// TwinCAT 3 PLC project SmartLiquidFillingSystem
// ProgramVersion: 3.1.4024.0
// libraries:
//   Tc2_Standard, * (Beckhoff Automation GmbH)
//   Tc2_System, * (Beckhoff Automation GmbH)
//   Tc3_Module, * (Beckhoff Automation GmbH)
// project tree:
//   DUTs/ E_LiquidType.TcDUT, E_StationState.TcDUT, ST_Bottle.TcDUT
//   GVLs/ GVL_References.TcGVL
//   / PlcTask.TcTTO
//   POUs/ FB_HoneyFill.TcPOU, FB_SodaFill.TcPOU, FB_StationController.TcPOU, FB_WaterFill.TcPOU, F_StrategyFunction.TcPOU, I_FillingStrategy.TcIO, MAIN.TcPOU
// (motion and I/O tree: see PLC project instructions_practice)
// real-time tasks:
//   TASK PlcTask: cycle T#10ms, priority 20, ADS port 350
//   TASK PlcTask1: cycle T#10ms, priority 22, ADS port 351
//   TASK PlcTask2: cycle T#10ms, priority 21, ADS port 352
//   TASK PlcTask3: cycle T#10ms, priority 23, ADS port 353

CONFIGURATION SmartLiquidFillingSystem
    RESOURCE PLC ON TwinCAT3
        TASK PlcTask(INTERVAL := T#10ms, PRIORITY := 23);
        PROGRAM MAIN WITH PlcTask : MAIN;
    END_RESOURCE
END_CONFIGURATION

// ---- DUTs/E_LiquidType.TcDUT
{attribute 'qualified_only'}
{attribute 'strict'}
TYPE E_LiquidType :
(
	WATER := 0,
	HONEY,
	SODA
);
END_TYPE

// ---- DUTs/E_StationState.TcDUT
{attribute 'qualified_only'}
{attribute 'strict'}
TYPE E_StationState :
(
	IDLE := 0,
	DETECTION,
	FILLING,
	COMPLETE,
	ERROR
);
END_TYPE

// ---- DUTs/ST_Bottle.TcDUT
TYPE ST_Bottle :
STRUCT
	nId  : DINT ;
	fCurrentLevel : REAL;
	fTargetLevel : REAL;
	eLiquidType : E_LiquidType;
END_STRUCT
END_TYPE

// ---- GVLs/GVL_References.TcGVL
{attribute 'qualified_only'}
VAR_GLOBAL
    g_fbHoneyFill : FB_HoneyFill;
    g_fbSodaFill  : FB_SodaFill;
    g_fbWaterFill : FB_WaterFill;
END_VAR

// ---- POUs/I_FillingStrategy.TcIO
INTERFACE I_FillingStrategy

METHOD ExecuteFill : BOOL
VAR_INPUT
	stBottle : REFERENCE TO ST_Bottle;
END_VAR
END_METHOD

END_INTERFACE

// ---- POUs/MAIN.TcPOU
PROGRAM MAIN
VAR
	bStart : BOOL;
	
	stBottle1 : ST_Bottle := (nId := 101, fTargetLevel := 70, eLiquidType := E_LiquidType.HONEY);
	stBottle2 : ST_Bottle := (nId := 102, fTargetLevel := 85, eLiquidType := E_LiquidType.SODA);
	stBottle3 : ST_Bottle := (nId := 103, fTargetLevel := 90, eLiquidType := E_LiquidType.WATER);
	
	
	fbStationController1 : FB_StationController;
	fbStationController2: FB_StationController;
	fbStationController3 : FB_StationController;
	
	
END_VAR

IF bStart THEN
	fbStationController1(stBottle := stBottle1);
	fbStationController2(stBottle := stBottle2);
	fbStationController3(stBottle := stBottle3);
	bStart := FALSE;
END_IF

END_PROGRAM

// ---- POUs/FB_StationController.TcPOU
FUNCTION_BLOCK FB_StationController

VAR_IN_OUT
	stBottle : ST_Bottle;
END_VAR
VAR
	iFillingStrategy : I_FillingStrategy;
	eStationState : E_StationState;
	nCompleteCount : DINT;
	nDefectCount : DINT;
END_VAR

IF  __ISVALIDREF(stBottle) THEN
	CASE eStationState OF
	E_StationState.IDLE:
		eStationState := E_StationState.DETECTION;
	
	E_StationState.DETECTION:
	iFillingStrategy := F_StrategyFunction(stBottle);
	IF iFillingStrategy <> 0 THEN
		eStationState := E_StationState.FILLING;
	ELSE
		eStationState := E_StationState.ERROR;
	END_IF
	
	E_StationState.FILLING:
	IF iFillingStrategy <> 0 THEN
		IF iFillingStrategy.ExecuteFill(stBottle) THEN
			eStationState := E_StationState.COMPLETE;
		END_IF
	END_IF
	
	E_StationState.COMPLETE:
	IF stBottle.fCurrentLevel = stBottle.fTargetLevel THEN
		nCompleteCount := nCompleteCount + 1;
	ELSE
		nDefectCount := nDefectCount + 1;
	END_IF
	eStationState := E_StationState.IDLE;
	
	E_StationState.ERROR:
	
	END_CASE
END_IF

END_FUNCTION_BLOCK

// ---- POUs/F_StrategyFunction.TcPOU
FUNCTION F_StrategyFunction : I_FillingStrategy
VAR_INPUT
	stBottle : REFERENCE TO ST_Bottle;
END_VAR

CASE stBottle.eLiquidType OF
	E_LiquidType.HONEY:
	F_StrategyFunction := GVL_References.g_fbHoneyFill ;
	
	E_LiquidType.SODA:
	F_StrategyFunction := GVL_References.g_fbSodaFill;
	
	E_LiquidType.WATER:
	F_StrategyFunction := GVL_References.g_fbWaterFill;
END_CASE

END_FUNCTION

// ---- POUs/FB_HoneyFill.TcPOU
FUNCTION_BLOCK FB_HoneyFill IMPLEMENTS I_FillingStrategy

VAR
END_VAR

{warning 'add method implementation '}
METHOD ExecuteFill : BOOL
VAR_INPUT
	stBottle: REFERENCE TO ST_Bottle;
END_VAR
VAR CONSTANT
	cFILLING_SPEED : REAL := 2;
END_VAR
IF __ISVALIDREF(stBottle) THEN
	IF stBottle.fCurrentLevel >= stBottle.fTargetLevel THEN
		ExecuteFill := TRUE;
	ELSE
		stBottle.fCurrentLevel := stBottle.fCurrentLevel + cFILLING_SPEED;
		ExecuteFill := FALSE;
	END_IF
END_IF
END_METHOD

END_FUNCTION_BLOCK

// ---- POUs/FB_SodaFill.TcPOU
FUNCTION_BLOCK FB_SodaFill IMPLEMENTS I_FillingStrategy
VAR_INPUT
END_VAR
VAR_OUTPUT
END_VAR
VAR
END_VAR

{warning 'add method implementation '}
METHOD ExecuteFill : BOOL
VAR_INPUT
	stBottle : REFERENCE TO ST_Bottle;
END_VAR

VAR CONSTANT
	cFILLING_SPEED: REAL:= 5;
END_VAR
IF __ISVALIDREF(stBottle) THEN
	IF stBottle.fCurrentLevel >= stBottle.fTargetLevel THEN
		ExecuteFill := TRUE;
	ELSE
		stBottle.fCurrentLevel := stBottle.fCurrentLevel + cFILLING_SPEED;
		ExecuteFill := FALSE;
	END_IF
END_IF
END_METHOD

END_FUNCTION_BLOCK

// ---- POUs/FB_WaterFill.TcPOU
FUNCTION_BLOCK FB_WaterFill IMPLEMENTS I_FillingStrategy
VAR_INPUT
END_VAR
VAR_OUTPUT
END_VAR
VAR
END_VAR

{warning 'add method implementation '}
METHOD ExecuteFill : BOOL
VAR_INPUT
	stBottle : REFERENCE TO ST_Bottle;
END_VAR

VAR CONSTANT
	cFILLING_SPEED: REAL := 10;
END_VAR
IF __ISVALIDREF(stBottle) THEN
	IF stBottle.fCurrentLevel >= stBottle.fTargetLevel THEN
		ExecuteFill := TRUE;
	ELSE
		stBottle.fCurrentLevel := stBottle.fCurrentLevel + cFILLING_SPEED;
		ExecuteFill := FALSE;
	END_IF
END_IF
END_METHOD

END_FUNCTION_BLOCK
